INTERFACE I_Device

METHOD Disable : bool
VAR_INPUT
END_VAR
END_METHOD

METHOD Enable : bool
VAR_INPUT
END_VAR
END_METHOD

METHOD Init : bool
VAR_INPUT
END_VAR
END_METHOD

METHOD Update : bool
VAR_INPUT
END_VAR
END_METHOD

END_INTERFACE

(* stored: Version 1.1.0.1
   Itf I_Device: Id {22acd9b2-801d-4255-af02-aa917c343cb7}
   Method Disable: Id {c1885dec-47ae-4f67-82bb-b5f267a6bb3b}
   Method Enable: Id {bb68bec4-22cd-4c90-90fd-577cff0dc9aa}
   Method Init: Id {586eeb72-004f-478a-90e1-1dfc38e6e530}
   Method Update: Id {8cb957b7-715c-48fb-8e7d-4bafd46d9bbc} *)
